TYPE ST_TransportMappingStationBuffer :
STRUCT
	{attribute 'OPC.UA.DA.Description' := 'Dummy (for making struct visible on OPC UA'}
	Dummy						: BOOL;

END_STRUCT
END_TYPE

(* stored: Version 1.1.0.1, ProductVersion 3.1.4024.5
   DUT ST_TransportMappingStationBuffer: Id {a0f66c74-d2db-43cb-b0f2-6958703992a0} *)
